// TIA Portal V20 export
// export: Created 2025-12-01T14:57:16.7301365Z, ExportSetting None, DisplayName Totally Integrated Automation Portal, DisplayVersion V20 Update 3, DisplayName TIA Portal Openness, DisplayVersion V20 Update 3, DisplayName TIA Portal Version Control Interface, DisplayVersion V20 Update 3, DisplayName STEP 7 Professional, DisplayVersion V20 Update 3, DisplayName STEP 7 Safety, DisplayVersion V20 Update 2, DisplayName WinCC Basic/Comfort/Advanced, DisplayVersion V20 Update 3, DisplayName WinCC Professional, DisplayVersion V20 Update 3, DisplayName WinCC Unified, DisplayVersion V20 Update 3
DATA_BLOCK "DB901_Estado_Zonas"   // DB901
{ S7_Optimized_Access := 'FALSE' }
AUTHOR : GENERAL
NAME : 20160413
VERSION : 3.1
// stored: AutoNumber false
   VAR RETAIN
      Maximo : Int := 100;   // Maximo Numero de Zonas
      Longitud : Int := 10;   // Tamaño de la Estructura de la Zona
      Offset : Int := 6;   // Offset de la Zona Numero 0
      EstadoZona { S7_SetPoint := 'True'} : Array[0.."CTE_MaxDispositivos"] of "UDT_EstadoZonaDispositivo";   // Zona de InterCambio de Datos con la Pantalla
   END_VAR
BEGIN
END_DATA_BLOCK
